(*
SPDX-FileCopyrightText: © 2026 Oleksandr Tiutyk <trofimich@gmail.com>
SPDX-License-Identifier: MIT
License: https://opensource.org/license/mit
*)

{attribute 'no_explicit_call' := 'do not call this function block directly'}
FUNCTION_BLOCK DemoExceptionHandlingPolicy EXTENDS TOF_Core.Object IMPLEMENTS TOF_Core.IExceptionHandlingPolicy
VAR_STAT
	//! <summary>Class name shared by all instances of this function block.</summary>
	{attribute 'hide'} 
	_ClassName : STRING := __POUNAME();
END_VAR

{attribute 'monitoring' := 'call'}
PROPERTY ClassName : REFERENCE TO STRING
GET
ClassName REF= _ClassName;
END_GET
END_PROPERTY

METHOD HandleException : TOF_Core.EXCEPTION_REACTION
VAR_INPUT
	exception : TOF_Core.IReadOnlyException;
	handlingObject : TOF_Core.IObject;
END_VAR
VAR_IN_OUT CONSTANT
	failedMethodName : STRING(255);
END_VAR
VAR
	demoException : IDemoException;
END_VAR
IF __QUERYINTERFACE(exception, demoException) THEN
	IF demoException.IsCritical THEN
		HandleException := TOF_Core.EXCEPTION_REACTION.SET_ERROR_AND_STOP;
	ELSE
		HandleException := TOF_Core.EXCEPTION_REACTION.SET_ERROR_AND_CONTINUE;
	END_IF
ELSE
	HandleException := TOF_Core.EXCEPTION_REACTION.SET_ERROR_AND_CONTINUE;
END_IF
END_METHOD

{attribute 'monitoring' := 'call'}
PROPERTY NamespaceName : REFERENCE TO STRING
GET
NamespaceName REF= CurrentNamespace.Name;
END_GET
END_PROPERTY

{attribute 'monitoring' := 'call'}
PROPERTY SelfSize : ULINT
GET
SelfSize := XSIZEOF(THIS^);
END_GET
END_PROPERTY

END_FUNCTION_BLOCK

(* stored: Version 1.1.0.1
   POU DemoExceptionHandlingPolicy: Id {c8288e63-0e66-4103-9ccf-5f7fe2e64839}, SpecialFunc None
   Property ClassName: Id {5f3d7f4b-db7b-473b-85f8-e9db3a59fd50}
   Get Get: Id {71703894-3bec-4ef1-88ec-919edbb71256}
   Method HandleException: Id {706f7f36-3413-49df-a7e7-8bbf8641a15d}
   Property NamespaceName: Id {33ae224c-325a-4b53-b26d-0997bf389202}
   Get Get: Id {fddebf50-b83f-4637-ba06-c017922efe20}
   Property SelfSize: Id {59668ee5-29ef-47bc-a58d-600fbc70e34c}
   Get Get: Id {96a00cc5-107c-476c-8923-16b68345967c} *)
